FUNCTION ByteArrayToReal : REAL
VAR_INPUT
	msg : CANQUEUE;
	pos : INT;
END_VAR
VAR_OUTPUT
	output : REAL;
END_VAR
VAR
	tmp: ARRAY[0..3] OF USINT;
	pt : POINTER TO REAL;
	i : INT;
END_VAR

FOR i := 0 TO 3 DO
	tmp[i] := msg.data[i+pos];
END_FOR
pt := ADR(tmp);
output := pt^;

END_FUNCTION

(* stored: Version 1.1.0.1, ProductVersion 3.1.4024.9
   POU ByteArrayToReal: Id {06c82136-d46e-41ad-b331-c03f2b4069b7}, SpecialFunc None *)
